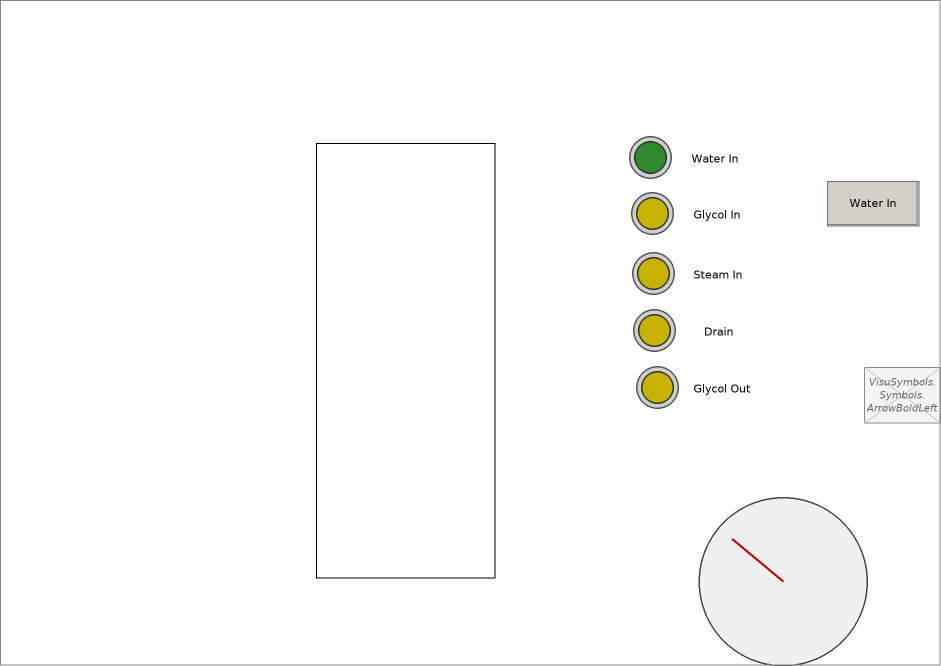
VISUALIZATION FermenterControl  // 941x666
    Rectangle (316,143 179x435)
    Lamp1 (624,133 53x49), variable: SFC.WaterIn, style: Lamp-Lamp1-Green
    Label (677,145 76x28), "Water In"
    Label (679,201 76x28), "Glycol In"
    Lamp1 (626,189 53x49), variable: SFC.GlycolIn, style: Lamp-Lamp1-Yellow
    Label (680,261 76x28), "Steam In"
    Lamp1 (627,249 53x49), variable: SFC.SteamIn, style: Lamp-Lamp1-Yellow
    Label (681,318 76x28), "Drain"
    Lamp1 (628,306 53x49), variable: SFC.Drain, style: Lamp-Lamp1-Yellow
    Label (684,375 76x28), "Glycol Out"
    Lamp1 (631,363 53x49), variable: SFC.GlycolOut, style: Lamp-Lamp1-Yellow
    Meter180 (651,497 264x169), value: SFC.Temp, style: Meter-Meter180-Gray, scale format: %.1f, scale 0..100
    Button (827,181 92x45), "Water In"
        OnMouseUp: toggle SFC.WaterIn
    Image (864,367 77x56), image: VisuSymbols.Symbols.ArrowBoldLeft
END_VISUALIZATION

(* stored: Version 1.1.0.1, ProductVersion 3.1.4024.12
   Visu FermenterControl: Id {d9033618-612d-48e6-b57a-dd52f264ebb0} *)
